TYPE ST_GCSingleProcessStageTimings :
STRUCT
	Prepare : ST_GCSingleProcessStageTiming;
	LiftReady : ST_GCSingleProcessStageTiming;
	SpinAlign : ST_GCSingleProcessStageTiming;
	ConcurrentProcessEntry : ST_GCSingleProcessStageTiming;
	SpinRampUp : ST_GCSingleProcessStageTiming;
	ProcessHold : ST_GCSingleProcessStageTiming;
	ConcurrentProcessExit : ST_GCSingleProcessStageTiming;
	SpinStandby : ST_GCSingleProcessStageTiming;
END_STRUCT
END_TYPE

(* stored: Version 1.1.0.1, ProductVersion 3.1.4026.18
   DUT ST_GCSingleProcessStageTimings: Id {1154e4ac-02fd-42a5-8e48-5143d0c00986} *)
